(* IEC 61131-3 sources: plc-agent/tests/fixtures/p3_broken, 2 files *)

(* ---- Broken.st ---- *)
FUNCTION_BLOCK FB_Broken
VAR_INPUT
    Fault : BOOL
END_VAR
END_FUNCTION_BLOCK

(* ---- Good.st ---- *)
FUNCTION_BLOCK FB_Healthy
VAR_OUTPUT
    Ready : BOOL;
END_VAR
Ready := TRUE;
END_FUNCTION_BLOCK
